(* Logix 5000 project; controller cal1632 1756-L62 rev 16.20; software revision 16.05; part 51 of 61 *)
(* tags used below, declared in another part *)
   di_request_move_a_to_doff : BOOL;
   di_request_move_a_to_run : BOOL;
   di_request_move_b_to_doff : BOOL;
   di_request_move_b_to_run : BOOL;
   FAULT : BOOL;
   HMI : BOOL;
   IN_ai_lc01 : ALIAS FOR Local:3:I.Ch2Data;
   p01_recipe_active : recipe;
   p01r02 : routine;
   p01r09_pb_global_reset : BOOL;
   p29_ai_radius : REAL;
   p29_ai_wa_amps : REAL;
   p29_ai_wa_dia_ft : REAL;
   p29_ai_wa_hz : REAL;
   p29_ai_wa_rpm : REAL;
   p29_ai_wa_speed : REAL;
   p29_ai_wa_torque : REAL;
   p29_ai_wb_amps : REAL;
   p29_ai_wb_dia_ft : REAL;
   p29_ai_wb_hz : REAL;
   p29_ai_wb_rpm : REAL;
   p29_ai_wb_speed : REAL;
   p29_ai_wb_torque : REAL;
   p29_ai_wdr_dia_in : REAL;
   p29_ai_wdr_lc : REAL;
   p29_ai_wdr_turret_amps : REAL;
   p29_ai_wdr_turret_hz : REAL;
   p29_ai_wdr_turret_speed : REAL;
   p29_ao_wa_torque_ref : REAL;
   p29_ao_wb_torque_ref : REAL;
   p29_di_wa_brake : BOOL;
   p29_di_wa_motor : BOOL;
   p29_di_wb_brake : BOOL;
   p29_di_wb_motor : BOOL;
   p29_di_wdr_a : BOOL;
   p29_di_wdr_a_core_size : BOOL;
   p29_di_wdr_a_reset_core : BOOL;
   p29_di_wdr_a_start : BOOL;
   p29_di_wdr_a_stop : BOOL;
   p29_di_wdr_b_core_size : BOOL;
   p29_di_wdr_b_reset_core : BOOL;
   p29_di_wdr_b_start : BOOL;
   p29_di_wdr_b_stop : BOOL;
   p29_di_wdr_index_fwd : BOOL;
   p29_di_wdr_jog : BOOL;
   p29_di_wdr_turret : acs800_di_normal;
   p29_di_wt_motor : BOOL;
   p29_dint_to_hmi : DINT[16];
   p29_param_lc_cal_factor : REAL;   // Winder Load Cell Calibration Factor Applied After Scaling
   p29_param_wa_gear_ratio : REAL;
   p29_param_wb_gear_ratio : REAL;
   p29_wa_footage_input_max : REAL;
   p29_wa_footage_input_min : REAL;
   p29_wa_footage_output_max : REAL;
   p29_wa_footage_output_min : REAL;
   p29_wb_footage_input_max : REAL;
   p29_wb_footage_input_min : REAL;
   p29_wb_footage_output_max : REAL;
   p29_wb_footage_output_min : REAL;
   p29_wda_status_word : INT;
   p29_wdb_status_word : INT;
   p29_wdr_diameter_input_max : REAL;
   p29_wdr_diameter_input_min : REAL;
   p29_wdr_diameter_output_max : REAL;
   p29_wdr_diameter_output_min : REAL;
   p29_wdr_lc_input_max : REAL;
   p29_wdr_lc_input_min : REAL;
   p29_wdr_lc_output_max : REAL;
   p29_wdr_lc_output_min : REAL;
   p29r01 : routine;
   p29r02 : routine;
   p29r02_fault_exists : BOOL;
   p29r02_tension_dev_max : REAL;
   p29r02_tension_dev_min : REAL;
   p29r02_timer_fault : TIMER[4];
   p29r02_timer_warning : TIMER[4];
   p29r02_unack_fault : BOOL;
   p29r02_unack_warning : BOOL;
   p29r02_wa_calc_torque_ref : REAL;
   p29r02_warning_exists : BOOL;
   p29r02_wb_calc_torque_ref : REAL;
   p29r02_winder_selection_dwell : TIMER;
   p29r03 : routine;
   p29r03_distance_to_core : REAL;
   p29r03_hz : SYS_SCP;
   p29r03_liner_wdr_lc_scp : SYS_SCP;
   p29r03_sample_timer : TIMER;
   p29r03_sensor_input : REAL;
   p29r03_timer_fault : TIMER[4];
   p29r03_timer_warning : TIMER[4];
   p29r03_unload : REAL;
   p29r03_wa_ave_tq : REAL;
   p29r03_wa_footage_scp : SYS_SCP;
   p29r03_wa_scaled_vfd_in : REAL;
   p29r03_wa_speed_fb : SYS_RPM_TO_SPEED;
   p29r03_wa_tq_ave_ctrl : CONTROL;
   p29r03_wa_tq_buffer : REAL[20];
   p29r03_wa_tq_fifo : CONTROL;
   p29r03_wb_ave_tq : REAL;
   p29r03_wb_footage_scp : SYS_SCP;
   p29r03_wb_scaled_vfd_in : REAL;
   p29r03_wb_speed_fb : SYS_RPM_TO_SPEED;
   p29r03_wb_tq_ave_ctrl : CONTROL;
   p29r03_wb_tq_buffer : REAL[20];
   p29r03_wb_tq_fifo : CONTROL;
   p29r03_wda_vfd_in_scaling : SYS_SCP;
   p29r03_wda_vfd_input_max : REAL;
   p29r03_wda_vfd_input_min : REAL;
   p29r03_wda_vfd_output_max : REAL;
   p29r03_wda_vfd_output_min : REAL;
   p29r03_wdb_vfd_in_scaling : SYS_SCP;
   p29r03_wdb_vfd_input_max : REAL;
   p29r03_wdb_vfd_input_min : REAL;
   p29r03_wdb_vfd_output_max : REAL;
   p29r03_wdb_vfd_output_min : REAL;
   p29r03_wdr_dia_sensor_scp : SYS_SCP;
   p29r04 : routine;
   p29r05 : routine;
   p29r06 : routine;
   p29r07 : routine;
   p29r08 : routine;
   p29r09 : routine;
   p29r10 : routine;
   p29r13_ai_wa_footage_ft : REAL;
   p29r13_ai_wb_footage_ft : REAL;
   p29r15 : routine;
   p29r15_wdra_active : BOOL;
   p29r16 : routine;
   p29r16_wdrb_active : BOOL;
   p29r17 : routine;
   p29r17_winder_a_avg_diam_inch : REAL;
   p29r18 : routine;
   p29r18_winder_b_avg_diam_inch : REAL;
   p29r20 : routine;

PROGRAM P29_Winder   (* main routine R01_Main *)
VAR
   abs_distance_to_move : REAL;   // Turret Absolute Distance to Move
   distance_to_move : REAL;   // Turret Distence to Move
   last_selected_position : REAL;   // Turret Last Selected Position
   p289_di_turret_in_position_bit_1 : BOOL;   // Winder Digital Input : Turret In Position Bit 1
   p289_di_turret_in_position_bit_2 : BOOL;   // Winder Digital Input : Turret In Position Bit 2
   p289_di_turret_in_position_bit_3 : BOOL;   // Winder Digital Input : Turret In Position Bit 3
   p29_param_tension_hi_limit : REAL := 250.0;   // Parameter Tension High Limit
   p29r15_drive_ok : BOOL;   // Winder A Drive Enable E-Stop Clear and Own Drive Healthy
   p29r16_drive_ok : BOOL;   // Winder B Drive Enable E-Stop Clear and Own Drive Healthy
   param_doff_position : REAL := 91.0;
   param_pos_db : REAL := 3.0;   // C: Turret Position Dead Band
   pb_jog_turret_rev : BOOL;   // HMI PB: Jog Turret Rev
   pos_hi_limit : REAL;   // Turret Position DB High Limit
   pos_hi_limit_temp : REAL;   // Turret Position High Limit Temp
   pos_lo_limit : REAL;   // Turret Position DB Low Limit
   pos_lo_limit_temp : REAL;   // Turret Position Low Limit Temp
   tmr_fwd_delay : TIMER := (PRE := 250);   // Turret Signal Dwell Timer
   tmr_ref_delay : TIMER := (PRE := 250);   // Turret Signal Dwell Timer
   turret_err_mod : REAL;   // Turret Shortest Path Error wrapped to 0..360
   turret_err_raw : REAL;   // Turret Shortest Path Raw error plus 540 offset
   turret_in_wda_run_position : BOOL;   // Turret In Winder A Run Position
   turret_in_wdb_run_position : BOOL;   // Turret In Winder B Run Position
   turret_index_active_last_scan : BOOL;   // Turret Index Active Last Scan
   turret_index_permissive : BOOL;   // Turret Index Permissive No Turret Drive Fault AND Neither Winder Requesting Run
   turret_request_reverse : BOOL;   // Turret Request Reverse Index
   turret_wa_pos_doff_request : BOOL;   // Turret Move to Winder A Doff Position Request
   turret_wa_pos_run_request : BOOL;   // Turret Move to Winder A Run Position
   turret_wb_pos_doff_request : BOOL;   // Turret Move to Winder B Doff Position Request
   turret_wb_pos_run_request : BOOL;   // Turret Move to Winder B Run Position
   wa_doff_pos : REAL;   // Turret Winder A Doff Position
   wa_run_position_high_limit : REAL;
   wa_run_position_low_limit : REAL;
   wb_doff_pos_tmp : REAL;   // Turret Temp Doff Position before MOD
   wb_doff_position : REAL;   // Turret Winder B Doff Position
   wb_run_position : REAL;   // Turret Winder B Run Position
   wb_run_position_high_limit : REAL;
   wb_run_position_low_limit : REAL;
   wb_run_position_tmp : REAL;   // Turret Temp Run Position before MOD
   winder_accel_rate : REAL := 25.0;
   winder_decel_rate : REAL := 25.0;
END_VAR

ROUTINE R01_Main   (* ladder *)
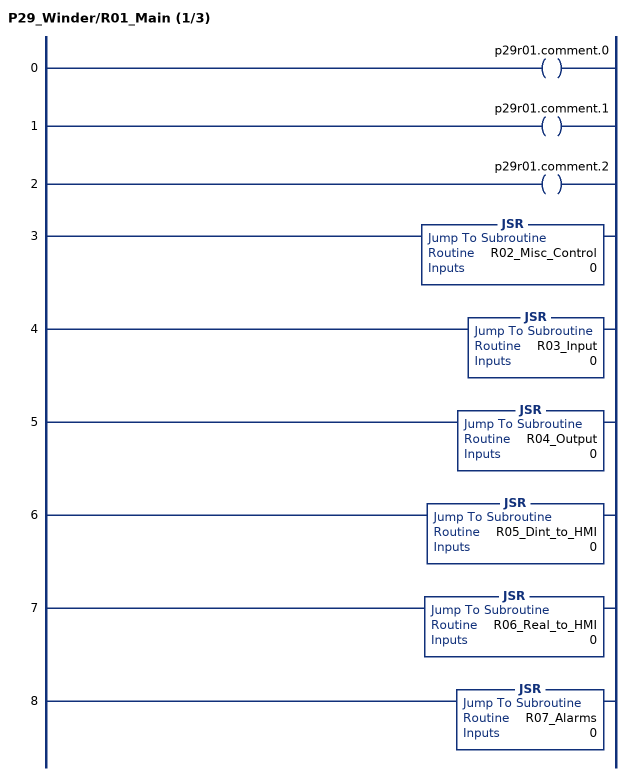
   0: OTE(p29r01.comment.0);
   1: OTE(p29r01.comment.1);
   2: OTE(p29r01.comment.2);
   3: JSR(R02_Misc_Control,0);
   4: JSR(R03_Input,0);
   5: JSR(R04_Output,0);
   6: JSR(R05_Dint_to_HMI,0);
   7: JSR(R06_Real_to_HMI,0);
   8: JSR(R07_Alarms,0);
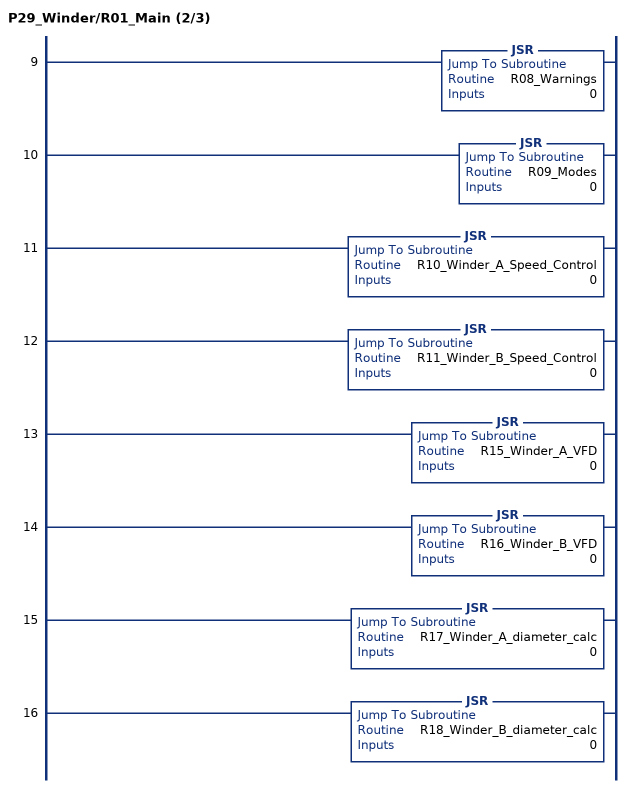
   9: JSR(R08_Warnings,0);
   10: JSR(R09_Modes,0);
   11: JSR(R10_Winder_A_Speed_Control,0);
   12: JSR(R11_Winder_B_Speed_Control,0);
   13: JSR(R15_Winder_A_VFD,0);
   14: JSR(R16_Winder_B_VFD,0);
   15: JSR(R17_Winder_A_diameter_calc,0);
   16: JSR(R18_Winder_B_diameter_calc,0);
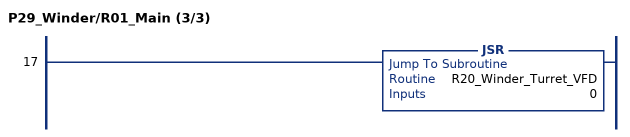
   17: JSR(R20_Winder_Turret_VFD,0);
END_ROUTINE

ROUTINE R02_Misc_Control   (* ladder *)
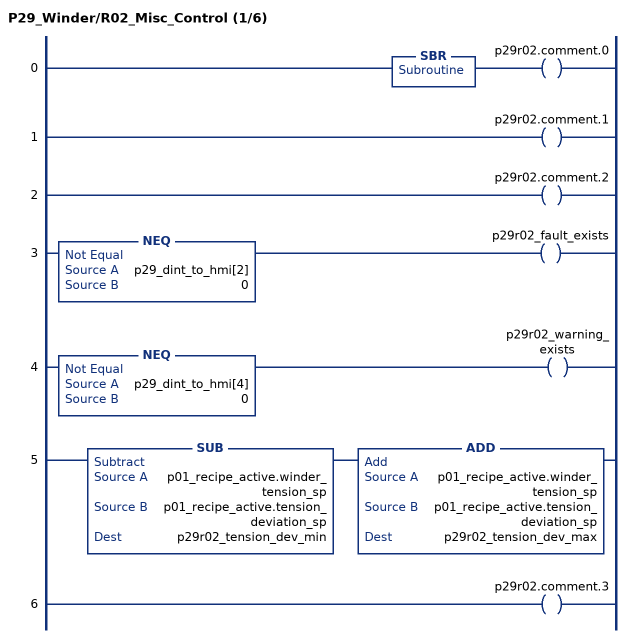
   0: SBR()OTE(p29r02.comment.0);
   1: OTE(p29r02.comment.1);
   2: OTE(p29r02.comment.2);
   3: NEQ(p29_dint_to_hmi[2],0)OTE(p29r02_fault_exists);
   4: NEQ(p29_dint_to_hmi[4],0)OTE(p29r02_warning_exists);
   5: SUB(p01_recipe_active.winder_tension_sp,p01_recipe_active.tension_deviation_sp,p29r02_tension_dev_min)ADD(p01_recipe_active.winder_tension_sp,p01_recipe_active.tension_deviation_sp,p29r02_tension_dev_max);
   6: OTE(p29r02.comment.3);
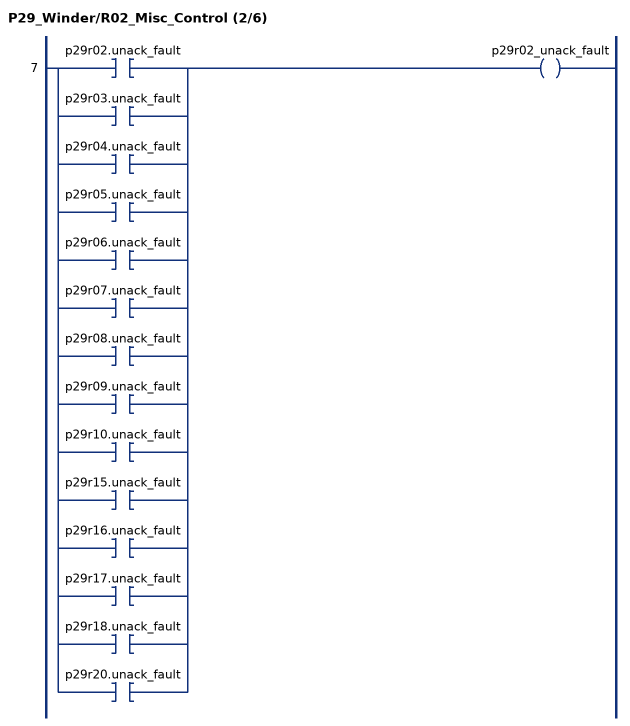
   7: [XIC(p29r02.unack_fault) ,XIC(p29r03.unack_fault) ,XIC(p29r04.unack_fault) ,XIC(p29r05.unack_fault) ,XIC(p29r06.unack_fault) ,XIC(p29r07.unack_fault) ,XIC(p29r08.unack_fault) ,XIC(p29r09.unack_fault) ,XIC(p29r10.unack_fault) ,XIC(p29r15.unack_fault) ,XIC(p29r16.unack_fault) ,XIC(p29r17.unack_fault) ,XIC(p29r18.unack_fault) ,XIC(p29r20.unack_fault) ]OTE(p29r02_unack_fault);
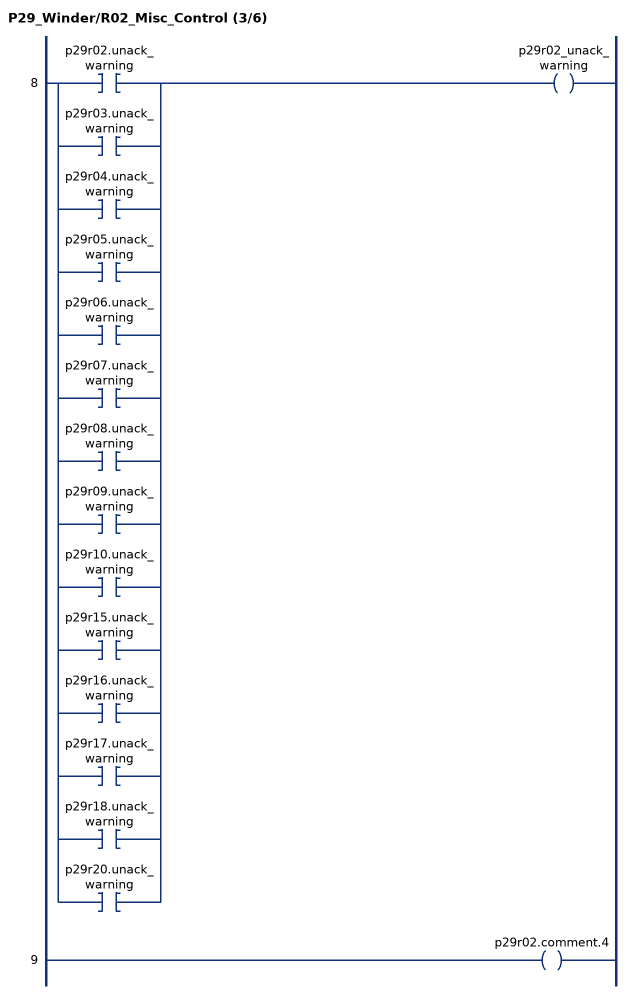
   8: [XIC(p29r02.unack_warning) ,XIC(p29r03.unack_warning) ,XIC(p29r04.unack_warning) ,XIC(p29r05.unack_warning) ,XIC(p29r06.unack_warning) ,XIC(p29r07.unack_warning) ,XIC(p29r08.unack_warning) ,XIC(p29r09.unack_warning) ,XIC(p29r10.unack_warning) ,XIC(p29r15.unack_warning) ,XIC(p29r16.unack_warning) ,XIC(p29r17.unack_warning) ,XIC(p29r18.unack_warning) ,XIC(p29r20.unack_warning) ]OTE(p29r02_unack_warning);
   9: OTE(p29r02.comment.4);
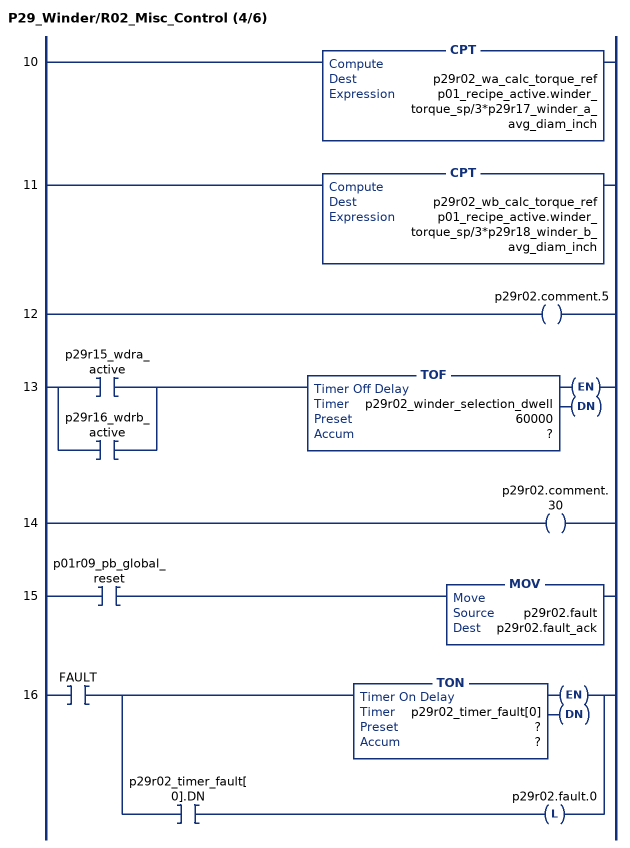
   10: CPT(p29r02_wa_calc_torque_ref,p01_recipe_active.winder_torque_sp/3*p29r17_winder_a_avg_diam_inch);
   11: CPT(p29r02_wb_calc_torque_ref,p01_recipe_active.winder_torque_sp/3*p29r18_winder_b_avg_diam_inch);
   12: OTE(p29r02.comment.5);
   13: [XIC(p29r15_wdra_active) ,XIC(p29r16_wdrb_active) ]TOF(p29r02_winder_selection_dwell,?,?);
   14: OTE(p29r02.comment.30);
   15: XIC(p01r09_pb_global_reset)MOV(p29r02.fault,p29r02.fault_ack);
   16: XIC(FAULT)[TON(p29r02_timer_fault[0],?,?) ,XIC(p29r02_timer_fault[0].DN) OTL(p29r02.fault.0) ];
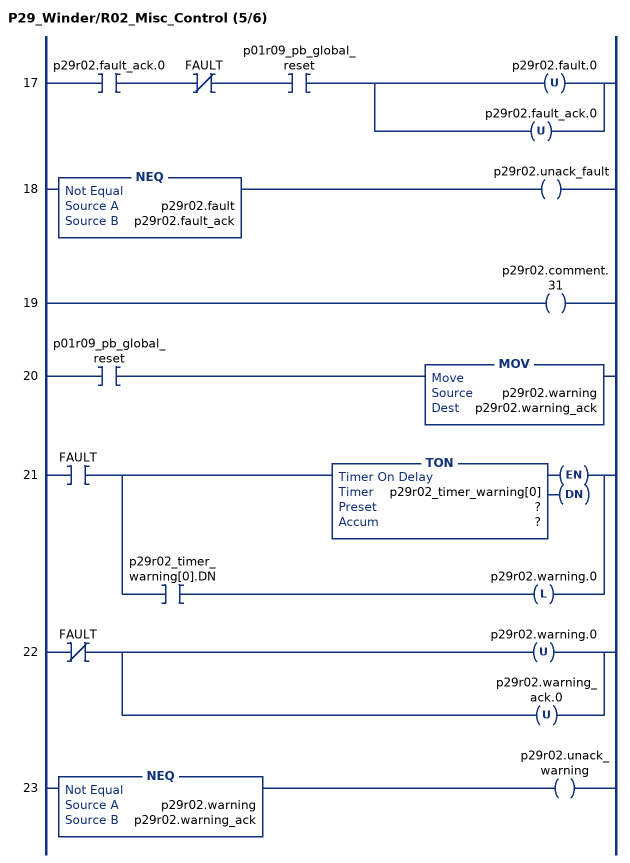
   17: XIC(p29r02.fault_ack.0)XIO(FAULT)XIC(p01r09_pb_global_reset)[OTU(p29r02.fault.0) ,OTU(p29r02.fault_ack.0) ];
   18: NEQ(p29r02.fault,p29r02.fault_ack)OTE(p29r02.unack_fault);
   19: OTE(p29r02.comment.31);
   20: XIC(p01r09_pb_global_reset)MOV(p29r02.warning,p29r02.warning_ack);
   21: XIC(FAULT)[TON(p29r02_timer_warning[0],?,?) ,XIC(p29r02_timer_warning[0].DN) OTL(p29r02.warning.0) ];
   22: XIO(FAULT)[OTU(p29r02.warning.0) ,OTU(p29r02.warning_ack.0) ];
   23: NEQ(p29r02.warning,p29r02.warning_ack)OTE(p29r02.unack_warning);
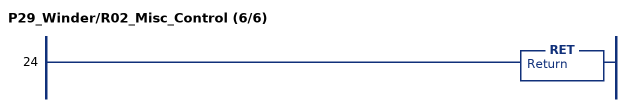
   24: RET();
END_ROUTINE

ROUTINE R03_Input   (* ladder *)
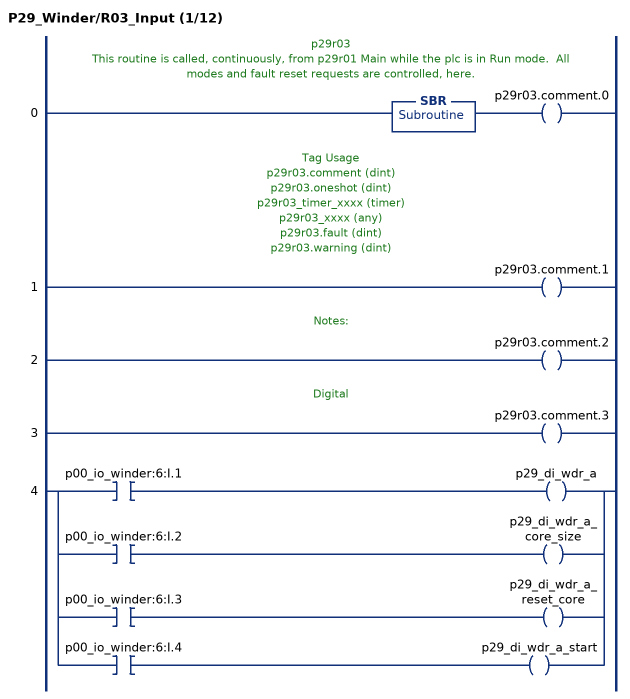
   // p29r03
   // This routine is called, continuously, from p29r01 Main while the plc is in Run mode.  All modes and fault reset requests are controlled, here.
   0: SBR()OTE(p29r03.comment.0);
   // Tag Usage
   // p29r03.comment (dint)
   // p29r03.oneshot (dint)
   // p29r03_timer_xxxx (timer)
   // p29r03_xxxx (any)
   // p29r03.fault (dint)
   // p29r03.warning (dint)
   1: OTE(p29r03.comment.1);
   // Notes:
   2: OTE(p29r03.comment.2);
   // Digital
   3: OTE(p29r03.comment.3);
   4: [XIC(p00_io_winder:6:I.1) OTE(p29_di_wdr_a) ,XIC(p00_io_winder:6:I.2) OTE(p29_di_wdr_a_core_size) ,XIC(p00_io_winder:6:I.3) OTE(p29_di_wdr_a_reset_core) ,XIC(p00_io_winder:6:I.4) OTE(p29_di_wdr_a_start) ];
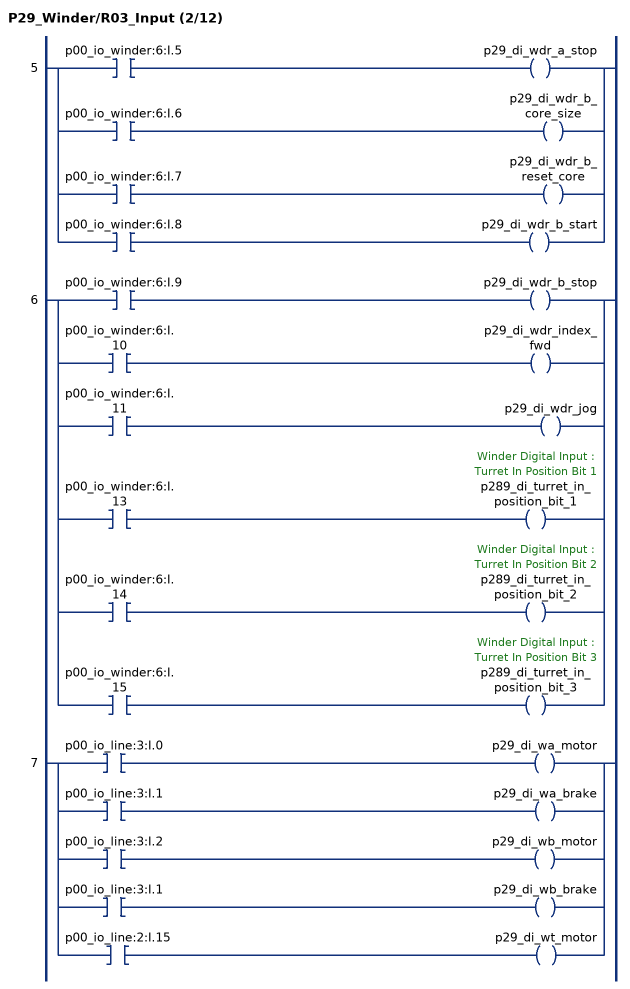
   5: [XIC(p00_io_winder:6:I.5) OTE(p29_di_wdr_a_stop) ,XIC(p00_io_winder:6:I.6) OTE(p29_di_wdr_b_core_size) ,XIC(p00_io_winder:6:I.7) OTE(p29_di_wdr_b_reset_core) ,XIC(p00_io_winder:6:I.8) OTE(p29_di_wdr_b_start) ];
   6: [XIC(p00_io_winder:6:I.9) OTE(p29_di_wdr_b_stop) ,XIC(p00_io_winder:6:I.10) OTE(p29_di_wdr_index_fwd) ,XIC(p00_io_winder:6:I.11) OTE(p29_di_wdr_jog) ,XIC(p00_io_winder:6:I.13) OTE(p289_di_turret_in_position_bit_1) ,XIC(p00_io_winder:6:I.14) OTE(p289_di_turret_in_position_bit_2) ,XIC(p00_io_winder:6:I.15) OTE(p289_di_turret_in_position_bit_3) ];
   7: [XIC(p00_io_line:3:I.0) OTE(p29_di_wa_motor) ,XIC(p00_io_line:3:I.1) OTE(p29_di_wa_brake) ,XIC(p00_io_line:3:I.2) OTE(p29_di_wb_motor) ,XIC(p00_io_line:3:I.1) OTE(p29_di_wb_brake) ,XIC(p00_io_line:2:I.15) OTE(p29_di_wt_motor) ];
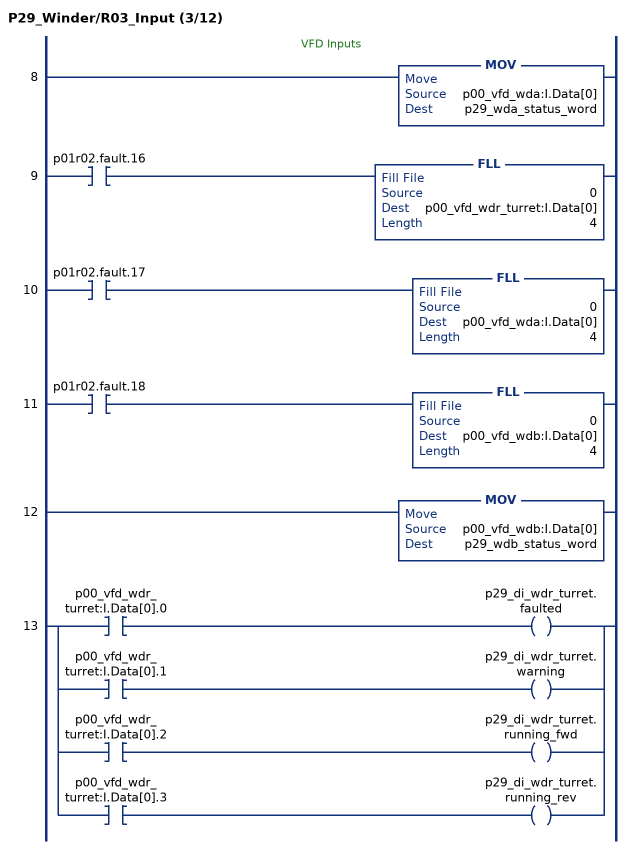
   // VFD Inputs
   8: MOV(p00_vfd_wda:I.Data[0],p29_wda_status_word);
   9: XIC(p01r02.fault.16)FLL(0,p00_vfd_wdr_turret:I.Data[0],4);
   10: XIC(p01r02.fault.17)FLL(0,p00_vfd_wda:I.Data[0],4);
   11: XIC(p01r02.fault.18)FLL(0,p00_vfd_wdb:I.Data[0],4);
   12: MOV(p00_vfd_wdb:I.Data[0],p29_wdb_status_word);
   13: [XIC(p00_vfd_wdr_turret:I.Data[0].0) OTE(p29_di_wdr_turret.faulted) ,XIC(p00_vfd_wdr_turret:I.Data[0].1) OTE(p29_di_wdr_turret.warning) ,XIC(p00_vfd_wdr_turret:I.Data[0].2) OTE(p29_di_wdr_turret.running_fwd) ,XIC(p00_vfd_wdr_turret:I.Data[0].3) OTE(p29_di_wdr_turret.running_rev) ];
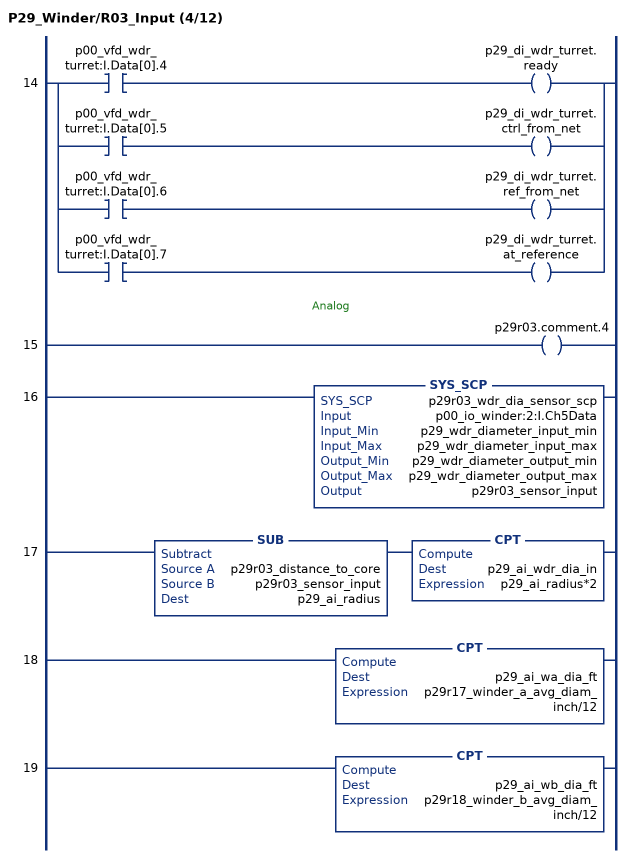
   14: [XIC(p00_vfd_wdr_turret:I.Data[0].4) OTE(p29_di_wdr_turret.ready) ,XIC(p00_vfd_wdr_turret:I.Data[0].5) OTE(p29_di_wdr_turret.ctrl_from_net) ,XIC(p00_vfd_wdr_turret:I.Data[0].6) OTE(p29_di_wdr_turret.ref_from_net) ,XIC(p00_vfd_wdr_turret:I.Data[0].7) OTE(p29_di_wdr_turret.at_reference) ];
   // Analog
   15: OTE(p29r03.comment.4);
   16: SYS_SCP(p29r03_wdr_dia_sensor_scp,p00_io_winder:2:I.Ch5Data,p29_wdr_diameter_input_min,p29_wdr_diameter_input_max,p29_wdr_diameter_output_min,p29_wdr_diameter_output_max,p29r03_sensor_input);
   17: SUB(p29r03_distance_to_core,p29r03_sensor_input,p29_ai_radius)CPT(p29_ai_wdr_dia_in,p29_ai_radius*2);
   18: CPT(p29_ai_wa_dia_ft,p29r17_winder_a_avg_diam_inch/12);
   19: CPT(p29_ai_wb_dia_ft,p29r18_winder_b_avg_diam_inch/12);
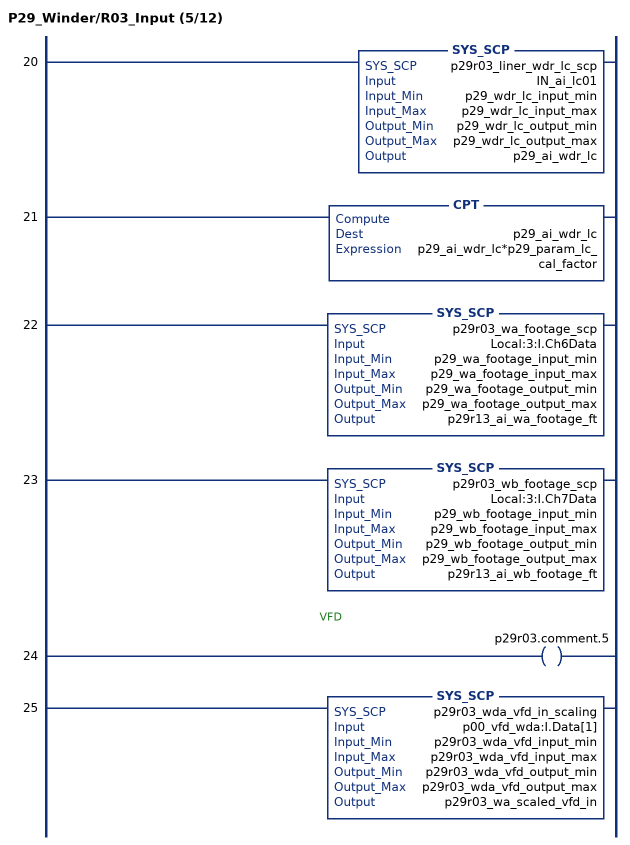
   20: SYS_SCP(p29r03_liner_wdr_lc_scp,IN_ai_lc01,p29_wdr_lc_input_min,p29_wdr_lc_input_max,p29_wdr_lc_output_min,p29_wdr_lc_output_max,p29_ai_wdr_lc);
   21: CPT(p29_ai_wdr_lc,p29_ai_wdr_lc*p29_param_lc_cal_factor);
   22: SYS_SCP(p29r03_wa_footage_scp,Local:3:I.Ch6Data,p29_wa_footage_input_min,p29_wa_footage_input_max,p29_wa_footage_output_min,p29_wa_footage_output_max,p29r13_ai_wa_footage_ft);
   23: SYS_SCP(p29r03_wb_footage_scp,Local:3:I.Ch7Data,p29_wb_footage_input_min,p29_wb_footage_input_max,p29_wb_footage_output_min,p29_wb_footage_output_max,p29r13_ai_wb_footage_ft);
   // VFD
   24: OTE(p29r03.comment.5);
   25: SYS_SCP(p29r03_wda_vfd_in_scaling,p00_vfd_wda:I.Data[1],p29r03_wda_vfd_input_min,p29r03_wda_vfd_input_max,p29r03_wda_vfd_output_min,p29r03_wda_vfd_output_max,p29r03_wa_scaled_vfd_in);
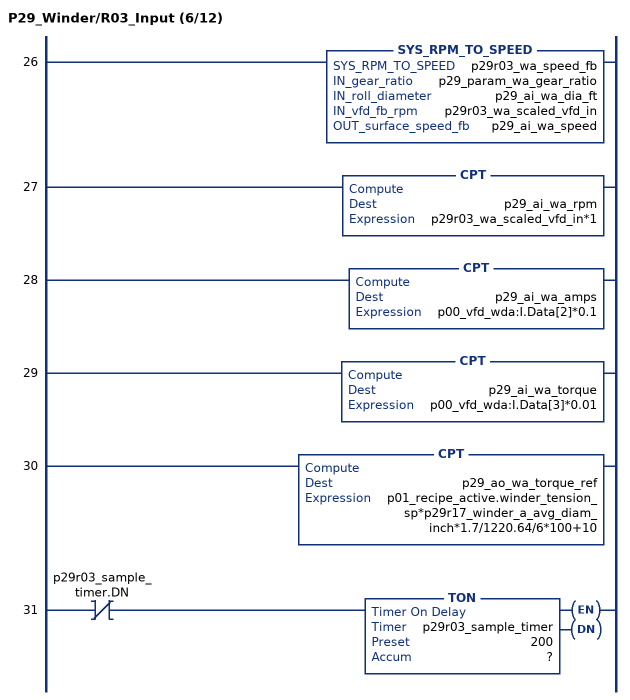
   26: SYS_RPM_TO_SPEED(p29r03_wa_speed_fb,p29_param_wa_gear_ratio,p29_ai_wa_dia_ft,p29r03_wa_scaled_vfd_in,p29_ai_wa_speed);
   27: CPT(p29_ai_wa_rpm,p29r03_wa_scaled_vfd_in*1);
   28: CPT(p29_ai_wa_amps,p00_vfd_wda:I.Data[2]*0.1);
   29: CPT(p29_ai_wa_torque,p00_vfd_wda:I.Data[3]*0.01);
   30: CPT(p29_ao_wa_torque_ref,p01_recipe_active.winder_tension_sp*p29r17_winder_a_avg_diam_inch*1.7/1220.64/6*100+10);
   31: XIO(p29r03_sample_timer.DN)TON(p29r03_sample_timer,?,?);
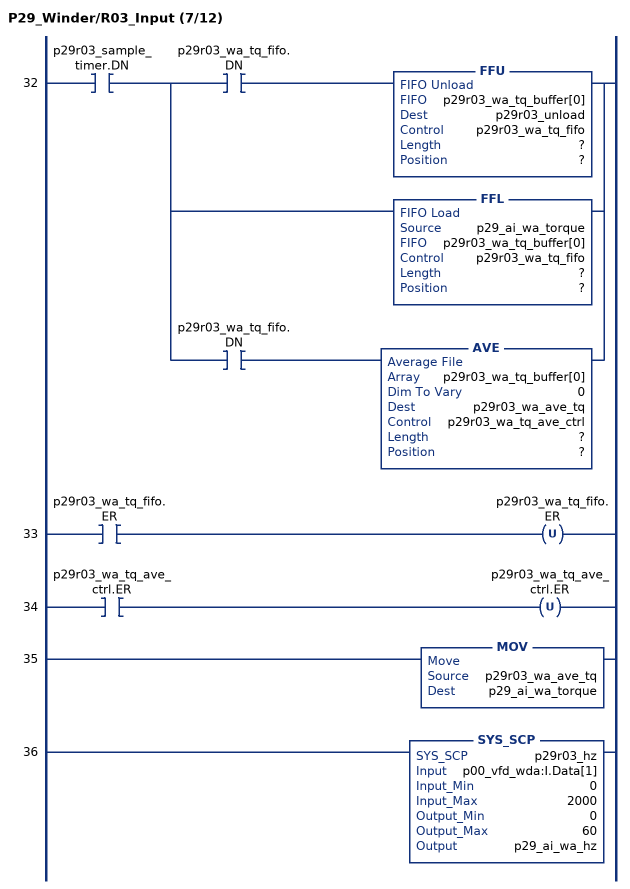
   32: XIC(p29r03_sample_timer.DN)[XIC(p29r03_wa_tq_fifo.DN) FFU(p29r03_wa_tq_buffer[0],p29r03_unload,p29r03_wa_tq_fifo,?,?) ,FFL(p29_ai_wa_torque,p29r03_wa_tq_buffer[0],p29r03_wa_tq_fifo,?,?) ,XIC(p29r03_wa_tq_fifo.DN) AVE(p29r03_wa_tq_buffer[0],0,p29r03_wa_ave_tq,p29r03_wa_tq_ave_ctrl,?,?) ];
   33: XIC(p29r03_wa_tq_fifo.ER)OTU(p29r03_wa_tq_fifo.ER);
   34: XIC(p29r03_wa_tq_ave_ctrl.ER)OTU(p29r03_wa_tq_ave_ctrl.ER);
   35: MOV(p29r03_wa_ave_tq,p29_ai_wa_torque);
   36: SYS_SCP(p29r03_hz,p00_vfd_wda:I.Data[1],0,2000,0,60,p29_ai_wa_hz);
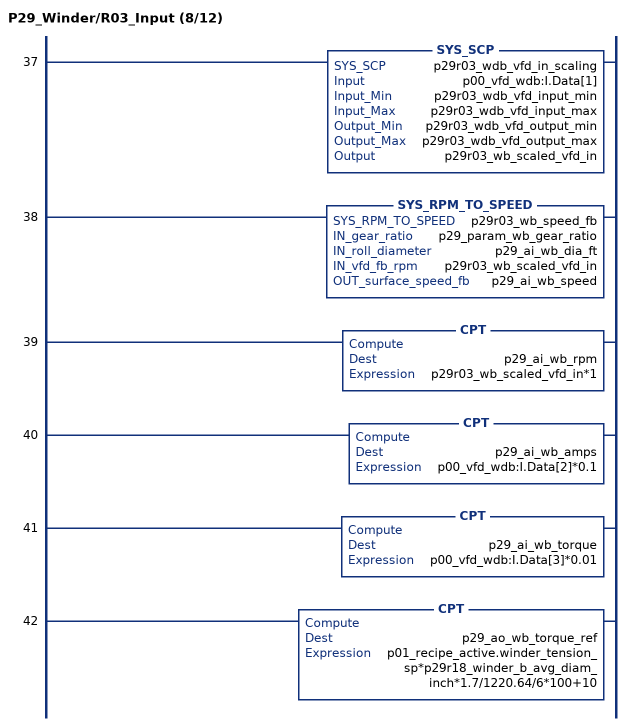
   37: SYS_SCP(p29r03_wdb_vfd_in_scaling,p00_vfd_wdb:I.Data[1],p29r03_wdb_vfd_input_min,p29r03_wdb_vfd_input_max,p29r03_wdb_vfd_output_min,p29r03_wdb_vfd_output_max,p29r03_wb_scaled_vfd_in);
   38: SYS_RPM_TO_SPEED(p29r03_wb_speed_fb,p29_param_wb_gear_ratio,p29_ai_wb_dia_ft,p29r03_wb_scaled_vfd_in,p29_ai_wb_speed);
   39: CPT(p29_ai_wb_rpm,p29r03_wb_scaled_vfd_in*1);
   40: CPT(p29_ai_wb_amps,p00_vfd_wdb:I.Data[2]*0.1);
   41: CPT(p29_ai_wb_torque,p00_vfd_wdb:I.Data[3]*0.01);
   42: CPT(p29_ao_wb_torque_ref,p01_recipe_active.winder_tension_sp*p29r18_winder_b_avg_diam_inch*1.7/1220.64/6*100+10);
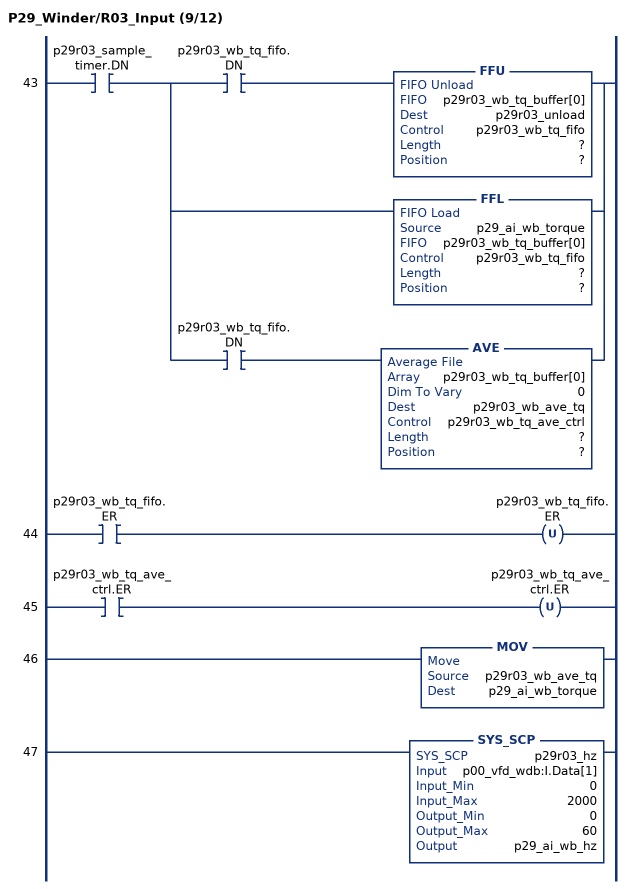
   43: XIC(p29r03_sample_timer.DN)[XIC(p29r03_wb_tq_fifo.DN) FFU(p29r03_wb_tq_buffer[0],p29r03_unload,p29r03_wb_tq_fifo,?,?) ,FFL(p29_ai_wb_torque,p29r03_wb_tq_buffer[0],p29r03_wb_tq_fifo,?,?) ,XIC(p29r03_wb_tq_fifo.DN) AVE(p29r03_wb_tq_buffer[0],0,p29r03_wb_ave_tq,p29r03_wb_tq_ave_ctrl,?,?) ];
   44: XIC(p29r03_wb_tq_fifo.ER)OTU(p29r03_wb_tq_fifo.ER);
   45: XIC(p29r03_wb_tq_ave_ctrl.ER)OTU(p29r03_wb_tq_ave_ctrl.ER);
   46: MOV(p29r03_wb_ave_tq,p29_ai_wb_torque);
   47: SYS_SCP(p29r03_hz,p00_vfd_wdb:I.Data[1],0,2000,0,60,p29_ai_wb_hz);
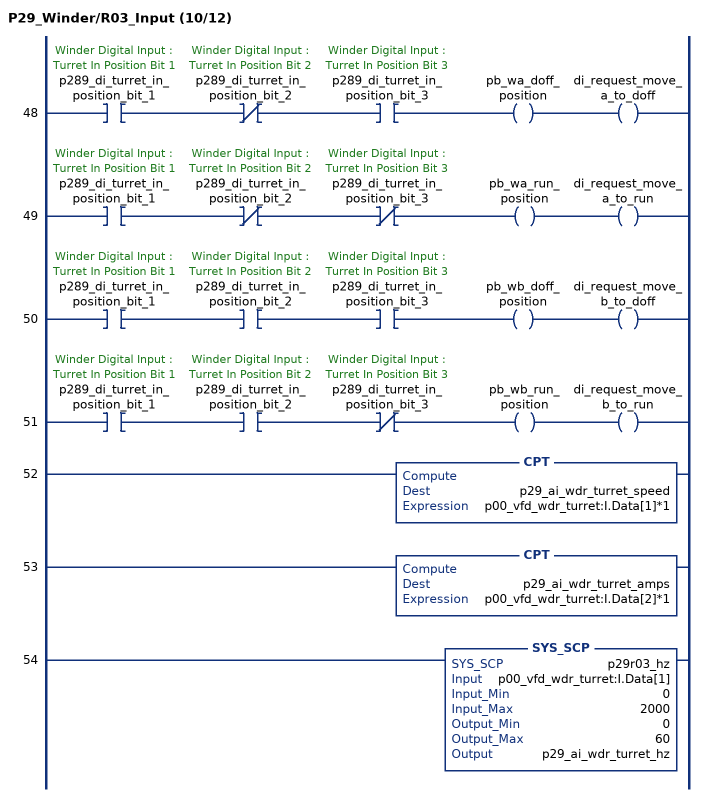
   48: XIC(p289_di_turret_in_position_bit_1)XIO(p289_di_turret_in_position_bit_2)XIC(p289_di_turret_in_position_bit_3)OTE(pb_wa_doff_position)OTE(di_request_move_a_to_doff);
   49: XIC(p289_di_turret_in_position_bit_1)XIO(p289_di_turret_in_position_bit_2)XIO(p289_di_turret_in_position_bit_3)OTE(pb_wa_run_position)OTE(di_request_move_a_to_run);
   50: XIC(p289_di_turret_in_position_bit_1)XIC(p289_di_turret_in_position_bit_2)XIC(p289_di_turret_in_position_bit_3)OTE(pb_wb_doff_position)OTE(di_request_move_b_to_doff);
   51: XIC(p289_di_turret_in_position_bit_1)XIC(p289_di_turret_in_position_bit_2)XIO(p289_di_turret_in_position_bit_3)OTE(pb_wb_run_position)OTE(di_request_move_b_to_run);
   52: CPT(p29_ai_wdr_turret_speed,p00_vfd_wdr_turret:I.Data[1]*1);
   53: CPT(p29_ai_wdr_turret_amps,p00_vfd_wdr_turret:I.Data[2]*1);
   54: SYS_SCP(p29r03_hz,p00_vfd_wdr_turret:I.Data[1],0,2000,0,60,p29_ai_wdr_turret_hz);
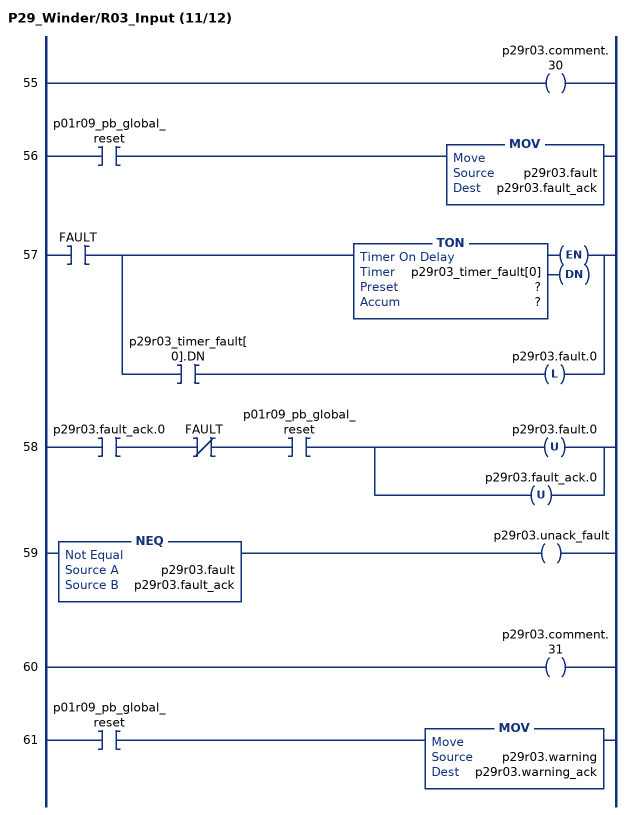
   55: OTE(p29r03.comment.30);
   56: XIC(p01r09_pb_global_reset)MOV(p29r03.fault,p29r03.fault_ack);
   57: XIC(FAULT)[TON(p29r03_timer_fault[0],?,?) ,XIC(p29r03_timer_fault[0].DN) OTL(p29r03.fault.0) ];
   58: XIC(p29r03.fault_ack.0)XIO(FAULT)XIC(p01r09_pb_global_reset)[OTU(p29r03.fault.0) ,OTU(p29r03.fault_ack.0) ];
   59: NEQ(p29r03.fault,p29r03.fault_ack)OTE(p29r03.unack_fault);
   60: OTE(p29r03.comment.31);
   61: XIC(p01r09_pb_global_reset)MOV(p29r03.warning,p29r03.warning_ack);
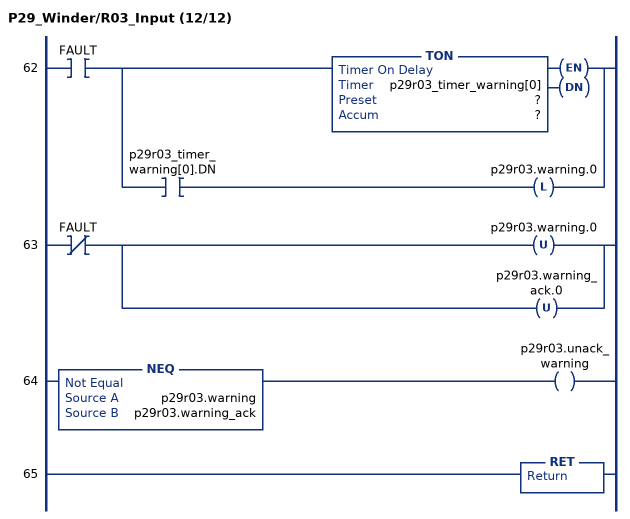
   62: XIC(FAULT)[TON(p29r03_timer_warning[0],?,?) ,XIC(p29r03_timer_warning[0].DN) OTL(p29r03.warning.0) ];
   63: XIO(FAULT)[OTU(p29r03.warning.0) ,OTU(p29r03.warning_ack.0) ];
   64: NEQ(p29r03.warning,p29r03.warning_ack)OTE(p29r03.unack_warning);
   65: RET();
END_ROUTINE
